FUNCTION write_bool_flag : BOOL
VAR_INPUT
	value : BOOL;
END_VAR
VAR
END_VAR

//Write bit register from PLC to Robot
//Flag to send to robot and indicate when the  system finish its process

write_bool_flag := FALSE;
Robot_UR5.UR_inputs.Bits.B0 := value;
Robot_UR5.UR_inputs.Bits.B1 := value;
Robot_UR5.UR_inputs.Bits.B2 := value;
write_bool_flag := TRUE;

END_FUNCTION

(* stored: Version 1.1.0.1, ProductVersion 3.1.4024.4
   POU write_bool_flag: Id {469482c1-564f-42de-8739-5ba175f383c9}, SpecialFunc None *)
